(* IEC 61131-3 sources: LASAL/Class/HWRtPostScan, 1 file *)

(* ---- HWRtPostScan.st ---- *)
(*!
<Class
	Name               = "HWRtPostScan"
	Revision           = "1.0"
	RealtimeTask       = "true"
	DefRealtimeIndex   = "1073741824"
	CyclicTask         = "false"
	BackgroundTask     = "false"
	Sigmatek           = "true"
	OSInterface        = "false"
	HighPriority       = "false"
	Automatic          = "false"
	UpdateMode         = "Prescan"
	IconPath           = ".\Class\HwControl\HwControl.ico"
	SharedCommandTable = "true"
	Objectsize         = "(660,120)">
	<Channels>
		<Server Name="ClassSvr" Visualized="false" Initialize="false" WriteProtected="true" Retentive="false"/>
		<Client Name="toHwControlBase" Required="true" Internal="false"/>
	</Channels>
	<RevDoku>
		<Owner Company="Sigmatek" Author="BleErn"/>
		<Dokumentation Revision="1.0" Date="08.02.2010" Author="BleErn" Company="Sigmatek" Description="Creation of class for implementation of HWRtPostScan"/>
	</RevDoku>
</Class>
*)
HWRtPostScan : CLASS
  //Servers:
	ClassSvr 	: SvrChCmd_DINT;
  //Clients:
	toHwControlBase 	: CltChCmd_HwControlBase;
  //Variables:
		RtTime 	: t_s_CyRtTime;
  //Functions:

	FUNCTION VIRTUAL GLOBAL RtWork
		VAR_INPUT
			EAX 	: UDINT;
		END_VAR
		VAR_OUTPUT
			state (EAX) 	: UDINT;
		END_VAR;
  //Tables:
	FUNCTION @STD
		VAR_OUTPUT
			ret_code	: CONFSTATES;
		END_VAR;
	FUNCTION GLOBAL TAB @CT_;
END_CLASS;

#pragma usingLtd HwControlBase

FUNCTION VIRTUAL GLOBAL HWRtPostScan::RtWork
	VAR_INPUT
		EAX 	: UDINT;
	END_VAR
	VAR_OUTPUT
		state (EAX) 	: UDINT;
	END_VAR

  toHwControlBase.UpdateRtPostScan();

	state := READY;

END_FUNCTION
